INTERFACE I_HostAsynchronousRpcHandlers

METHOD PUBLIC RegisterHandler
VAR_INPUT
	MethodName : T_MAXSTRING;
	Handler : I_AsynchronousRpcHandler;
END_VAR
END_METHOD

END_INTERFACE

(* stored: Version 1.1.0.1, ProductVersion 3.1.4026.13
   Itf I_HostAsynchronousRpcHandlers: Id {78bf5133-afc5-0ea6-1f61-79b4313bdee0}
   Method RegisterHandler: Id {1feda56d-fc6f-0a58-0484-aadd70f56a52} *)
